TYPE StepLog_Struct :
STRUCT
	step_number : DINT;
	created_at : LINT;
	program_name : STRING(80);
	extras_Srt : STRING(255) := '{}';
END_STRUCT
END_TYPE

(* stored: Version 1.1.0.1, ProductVersion 3.1.4026.13
   DUT StepLog_Struct: Id {14dda15e-6c8b-4a22-80d3-7b17bbdca453} *)
